PROGRAM MAIN
VAR
	my_counter : INT := 0;
	btn : BOOL;
	lmp : BOOL;
END_VAR

my_counter := my_counter + 2;

gvl.lamp_on := gvl.button_pressed;

END_PROGRAM

(* stored: Version 1.1.0.1, ProductVersion 3.1.4024.12
   POU MAIN: Id {31400cb4-b4cb-40c4-b7a1-915ff1e2cd27}, SpecialFunc None *)
